(*

.. <legal notes>

legal notes
=================
| SPDX-FileCopyrightText: © 2025 Oleksandr Tiutyk <trofimich@gmail.com>
| SPDX-License-Identifier: LGPL-3.0-only
| For details check: LGPL-3.0-only_

.. _LGPL-3.0-only: https://www.gnu.org/licenses/lgpl-3.0.en.html

.. </legal notes>

*)

INTERFACE INamedObject EXTENDS IObject

{attribute 'monitoring' := 'call'}
PROPERTY Name : WSTRING
GET
END_GET
END_PROPERTY

END_INTERFACE

(* stored: Version 1.1.0.1
   Itf INamedObject: Id {dd8cabbd-8ae8-4ca5-85c9-3758bf241bdb}
   Property Name: Id {d5712a44-804d-4034-89b5-de41f1b06d86}
   Get Get: Id {6cf39e17-2370-4943-9c4f-735bf1678b9c} *)
